TYPE U_OdriveSetAbsolutePositionBytes :
UNION
    stSetAbsolutePosition : ST_OdriveSetAbsolutePosition;
    aBytes : ARRAY[0..3] OF BYTE;
END_UNION
END_TYPE

(* stored: Version 1.1.0.1
   DUT U_OdriveSetAbsolutePositionBytes: Id {f9341c3f-5ddd-462b-900e-3af1480b55de} *)
